Fanuc KAREL source: kb00095.KL

-- PROVISIONAL review KL for V940-1; original PC SHA256 4f9f6588dd61d19eecbabec128e863581dc1d6f1bcd5b754f1b9e2925be4bf77
-- Incomplete behavior may be omitted. Consult companion uncertainty JSON. Do not deploy.
PROGRAM KB00095
%NOLOCKGROUP
BEGIN
  -- V9_ZERO_TABLE_METADATA_HINT layout=0002_ascii; no indexed target words; source/name/runtime held
  -- UNRESOLVED_PC offsets 5-12; opcodes 9D,23
  -- UNRESOLVED_PC offsets 17-24; opcodes 9D,23
  -- UNRESOLVED_PC offsets 29-38; opcodes 3F,75
  -- UNRESOLVED_PC offsets 43-50; opcodes 9D,23
  -- UNRESOLVED_PC offsets 55-85; opcodes 27,22,22,22,2A,22,31
  -- UNRESOLVED_PC offsets 90-94; opcodes 7F
END KB00095
